TYPE Coordonnees :
STRUCT
	X, Y, Z : LREAL;
END_STRUCT
END_TYPE

(* stored: Version 1.1.0.1, ProductVersion 3.1.4024.15
   DUT Coordonnees: Id {00172d99-4847-48df-9158-cbec50055615} *)
